FUNCTION_BLOCK FB_LoadCell_Sim IMPLEMENTS I_LoadCell
VAR_INPUT
END_VAR
VAR_OUTPUT
END_VAR
VAR
	bEnable : BOOL;
	fValue  : REAL;
	wStatus : WORD;
	// var Sim
	nState  		: INT;
	fSetpoint		: REAL := 1000000;//setpoint feedback speed Loadcell 
	tTimer			: TON; 
	bInit			: BOOL := TRUE;
END_VAR

CASE nState OF
	0: //init
		IF bInit THEN
			fValue := 0;
		END_IF
		nState := nState + 1;
	1://Loadcell Stop
		fValue := 0;
	
	10: // check have cup on loadcell
		IF bHaveLoad THEN
			nState := 20;
		END_IF
	20:
		fValue := fValue + fInvSpeed/fSetpoint;
		IF NOT bHaveLoad THEN
			nState := 10;
		END_IF
END_CASE
//check enable loadcell
IF (nState = 1) AND bEnable THEN
	tTimer(IN := FALSE);
	nState := 10;//Loadcell start
END_IF

PROPERTY fActWeight : REAL
GET
fActWeight := fValue;
END_GET
END_PROPERTY

METHOD NetMode : BOOL
VAR_INPUT
END_VAR
bEnable := true;
END_METHOD

METHOD Set_Zero : BOOL
VAR_INPUT
END_VAR
fValue := 0;
END_METHOD

PROPERTY Status : REAL
GET
Status := WORD_TO_REAL(wStatus);
END_GET
END_PROPERTY

END_FUNCTION_BLOCK

(* stored: Version 1.1.0.1, ProductVersion 3.1.4024.12
   POU FB_LoadCell_Sim: Id {3e911fc9-a1ad-4ef8-bcff-494fb39ecacb}, SpecialFunc None
   Property fActWeight: Id {2e7f61a7-07e3-4727-8fa9-99bc9e8be95c}
   Get Get: Id {f99bc1d7-d9af-49ca-9d42-202598be6d16}
   Method NetMode: Id {73ca5b07-5b39-4839-b99e-ea08226c9cd4}
   Method Set_Zero: Id {5e28bb37-6392-4580-b3d3-b1263d4d25fd}
   Property Status: Id {f9c681c7-8f0c-4832-8688-f20953bf4759}
   Get Get: Id {b8411849-765b-4608-b7b4-dc7c3fdb93fe} *)
